Universal Robots PolyScope program: CameraCalibrate.urp

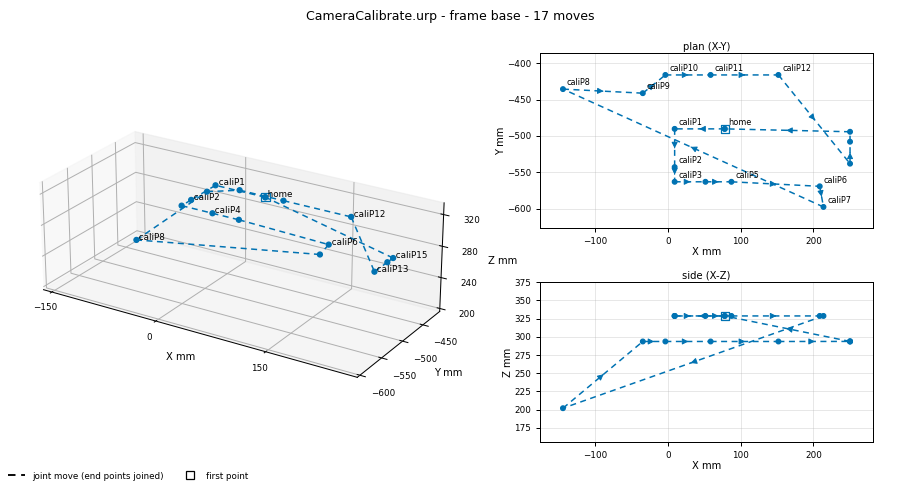
[picture p0: tool path of CameraCalibrate.urp in frame base, 17 of 17 moves have a stored position in this frame; points joined in program order, loops and branches not executed]
Program CameraCalibrate (installation=default directory=/programs/cam createdIn=5.19.0 lastSavedIn=5.15.1 robotSerialNumber=20245500285)
Calibrated DH parameters: a=[0.000097, -0.210459, -0.026602, 0.000137, 0.000078, 0]; d=[0.162601, 254.180657, -54.076236, -199.970743, 0.099615, 0.099684]; alpha=[1.569796, -0.001455, 0.001957, 1.570525, -1.571561, 0]; deltaTheta=[0, -1.053331, 8.839472, -1.50296, 0.000002, 0]
InitVariablesNode
Robot Program (runOnlyOnce=true)
  Script file /programs/cam/camera.script
    | def CameraOpenSock(ip, port=8888):
    |   socket_open(ip, port, "socker_camera")
    | end
    | 
    | 
    | def CameraCloseSock():
    |   socket_close("socker_camera")
    | end
    | 
    | 
    | def CameraSwitchOnline():
    |   socket_send_string("2\r", "socker_camera")
    |   ret = socket_read_string("socker_camera", suffix="\r")
    |   if (ret == "-1"):
    |     popup("CameraSwitchOnline Error", title="2.5D Camera", blocking=True)
    |   elif (ret == ""):
    |     popup("CameraSwitchOnline Error | Recv Data is None", title="2.5D Camera", blocking=True)
    |   end
    | end
    | 
    | 
    | def CameraStartCalibrate():
    |   socket_send_string("3\r", "socker_camera")
    |   ret = socket_read_string("socker_camera", suffix="\r")
    |   if (ret == "-1"):
    |     popup("CameraStartCalibrate Error", title="2.5D Camera", blocking=True)
    |   elif (ret == ""):
    |     popup("CameraStartCalibrate Error | Recv Data is None", title="2.5D Camera", blocking=True)
    |   end
    | end
    | 
    | def format03f(num):
    |   s = to_str(num)
    |   index = str_find(s, ".")
    |   if index != -1:
    |     ret = str_sub(s,0, index + 3)
    |     return ret
    |   else:
    |     return "rt"
    |   end
    | end
    | 
    | def CameraPackPose(pose):
    |   ret = ["", "", "", "", "", ""]
    |   pose[0] = pose[0] * 1000
    |   pose[1] = pose[1] * 1000
    |   pose[2] = pose[2] * 1000
    |   rpy = rotvec2rpy([pose[3], pose[4], pose[5]])
    |   ret[0] = format03f(pose[0])
    |   ret[1] = format03f(pose[1])
    |   ret[2] = format03f(pose[2])
    |   ret[3] = format03f(r2d(rpy[0]))
    |   ret[4] = format03f(r2d(rpy[1]))
    |   ret[5] = format03f(r2d(rpy[2]))
    |   i = 0
    |   out = ""
    |   while i < 6:
    |     out = str_cat(str_cat(out, ret[i]), ",")
    |     i = i + 1
    |   end
    | 
    |   return out
    | end
    | 
    | def CameraUnpackPose(text):
    |   ret = [0, 0, 0, 0, 0, 0, 0]
    |   i = 0
    |   index = 1
    |   while 1:
    |     index = str_find(text, ",")
    |     if index == -1:
    |       ret[i] = to_num(str_sub(text, 0))
    |     else:
    |       ret[i] = to_num(str_sub(text, 0, index))
    |     end
    |     text = str_sub(text, index+1)
    |     i=i+1
    |     if i > 6:
    |       break
    |     end
    |   end
    |   return ret
    | end
    | 
    | def CameraCalibrate(pose, num):
    | 
    |   pose1 = CameraPackPose(pose)
    |   sendStr = str_cat("", pose1)
    |   sendStr = str_cat("4,", sendStr)
    |   sendStr = str_cat(sendStr, to_str(num))
    |   sendStr = str_cat(sendStr, "\r")
    |   socket_send_string(sendStr, "socker_camera")
    |   ret = socket_read_string("socker_camera", suffix="\r")
    |   if (ret == "-1"):
    |     popup("CameraCalibrate Error", title="2.5D Camera", blocking=True)
    |   elif (ret == ""):
    |     popup("CameraCalibrate Error | Recv Data is None", title="2.5D Camera", blocking=True)
    |   end
    | end
    | 
    | 
    | def CameraEndCalibrate():
    |   socket_send_string("5\r", "socker_camera")
    |   ret = socket_read_string("socker_camera", suffix="\r")
    |   if (ret == "-1"):
    |     popup("CameraEndCalibrate Error", title="2.5D Camera", blocking=True)
    |   elif (ret == ""):
    |     popup("CameraEndCalibrate Error | Recv Data is None", title="2.5D Camera", blocking=True)
    |   end
    | end
    | 
    | 
    | def CameraGetCalibrateResult():
    | 
    |   socket_send_string("6\r")
    |   ret = socket_read_string("socker_camera", suffix="\r")
    |   if (ret == "-1"):
    |     popup("CameraGetCalibrateResult Error", title="2.5D Camera", blocking=True)
    |   elif (ret == ""):
    |     popup("CameraGetCalibrateResult Error | Recv Data is None", title="2.5D Camera", blocking=True)
    |   end
    | end
    | 
    | def CameraGetMarkPose():
    |   socket_send_string("1\r")
    |   ret = socket_read_string("socker_camera", suffix="\r")
    |   if (ret == "-1"):
    |     popup("CameraGetMarkPose Error", title="2.5D Camera", blocking=True)
    |   elif (ret == ""):
    |     popup("CameraGetMarkPose Error | Recv Data is None", title="2.5D Camera", blocking=True)
    |   else:
    |     result = CameraUnpackPose(ret)
    |     x = result[1] / 1000
    |     y = result[2] / 1000
    |     z = result[3] / 1000
    |     rx = d2r(result[4])
    |     ry = d2r(result[5])
    |     rz = d2r(result[6])
    |     rotvec2rpy = rpy2rotvec([rx, ry, rz])
    |     return [x, y, z, rotvec2rpy[0], rotvec2rpy[1], rotvec2rpy[2]]
    |   end
    | end
    | 
    | 
    | def CameraSaveTemplate(boardPose, tool=get_actual_tcp_pose()):
    |   # global CameraTemplate
    |   CameraTemplate = pose_trans(tool, boardPose)
    |   return CameraTemplate
    | end
    | 
    | def CameraTrsf(t, nT, p, tool=get_actual_tcp_pose()):
    |   trsf = pose_trans(pose_inv(t), p)
    |   ret = pose_trans(nT, trsf)
    |   return ret
    | end
  Script: CameraOpenSock("192.168.1.99", 8888)
  Script: CameraStartCalibrate()
  MoveJ speed 60 deg/s, acceleration 80 deg/s^2 (useActiveTCP=true) feature=Base
    Waypoint home: TCP in base x=78.162 y=-490.219 z=328.716 mm, rx=1.953 ry=2.4607 rz=0 rad; joints [83.356, -87.304, 111.233, -113.971, -90.025, 70.396] deg
    Script: CameraCalibrate(get_actual_tcp_pose(),1)
  MoveJ speed 60 deg/s, acceleration 80 deg/s^2 (useActiveTCP=true) feature=Base
    Waypoint caliP1: TCP in base x=9.395 y=-490.216 z=328.711 mm, rx=1.8055 ry=2.275 rz=0.262 rad; joints [71.893, -88.338, 111.523, -108.01, -74.336, 58.227] deg
    Script: CameraCalibrate(get_actual_tcp_pose(),2)
    Waypoint caliP2: TCP in base x=9.386 y=-542.747 z=328.724 mm, rx=1.8823 ry=2.3141 rz=0.4621 rad; joints [74.13, -79.525, 99.578, -96.524, -76.666, 60.977] deg
    Script: CameraCalibrate(get_actual_tcp_pose(),3)
    Waypoint caliP3: TCP in base x=9.395 y=-562.886 z=328.708 mm, rx=-1.9478 ry=-2.3477 rz=-0.4503 rad; joints [76.344, -75.67, 93.847, -91.652, -85.665, 65.265] deg
    Script: CameraCalibrate(get_actual_tcp_pose(),4)
    Waypoint caliP4: TCP in base x=51.659 y=-562.887 z=328.728 mm, rx=-1.9083 ry=-2.2531 rz=-0.2891 rad; joints [81.931, -75.392, 93.786, -93.635, -92.499, 72.966] deg
    Script: CameraCalibrate(get_actual_tcp_pose(),5)
    Waypoint caliP5: TCP in base x=87.316 y=-562.899 z=328.725 mm, rx=-1.8729 ry=-2.1767 rz=-0.1707 rad; joints [86.57, -74.564, 92.86, -93.637, -97.887, 79.191] deg
    Script: CameraCalibrate(get_actual_tcp_pose(),6)
    Waypoint caliP6: TCP in base x=208.594 y=-569.092 z=328.725 mm, rx=-1.7604 ry=-1.959 rz=0.1217 rad; joints [100.768, -67.818, 83.402, -84.689, -111.16, 98.788] deg
    Script: CameraCalibrate(get_actual_tcp_pose(),7)
    Waypoint caliP7: TCP in base x=213.728 y=-597.42 z=328.73 mm, rx=-1.7055 ry=-1.9272 rz=0.1003 rad; joints [100.941, -63.086, 76.071, -78.574, -112.507, 99.081] deg
    Script: CameraCalibrate(get_actual_tcp_pose(),8)
    Waypoint caliP8: TCP in base x=-143.969 y=-435.62 z=202.03 mm, rx=-0.4349 ry=2.6519 rz=0.5042 rad; joints [-95.138, -102.858, -115.737, -78.365, 106.879, -27.84] deg
    Script: CameraCalibrate(get_actual_tcp_pose(),9)
    Waypoint caliP9: TCP in base x=-34.347 y=-441.212 z=293.647 mm, rx=1.7983 ry=2.2001 rz=0.0566 rad; joints [63.83, -93.734, 124.614, -122.707, -72.812, 52.787] deg
    Script: CameraCalibrate(get_actual_tcp_pose(),10)
    Waypoint caliP10: TCP in base x=-3.351 y=-416.174 z=293.66 mm, rx=1.7423 ry=2.1705 rz=-0.1183 rad; joints [66.091, -98.263, 131.424, -133.489, -71.673, 55.418] deg
    Script: CameraCalibrate(get_actual_tcp_pose(),11)
    Waypoint caliP11: TCP in base x=58.77 y=-416.17 z=293.653 mm, rx=1.8028 ry=2.3259 rz=-0.352 rad; joints [78.661, -96.575, 131.561, -141.783, -87.034, 64.797] deg
    Script: CameraCalibrate(get_actual_tcp_pose(),12)
    Waypoint caliP12: TCP in base x=151.884 y=-416.164 z=293.638 mm, rx=-1.7862 ry=-2.419 rz=0.6473 rad; joints [96.807, -90.978, 126.971, -141.679, -109.249, 77.154] deg
    Script: CameraCalibrate(get_actual_tcp_pose(),13)
    Waypoint caliP13: TCP in base x=250.21 y=-538.008 z=293.739 mm, rx=-1.6396 ry=-2.0966 rz=0.2595 rad; joints [105.87, -68.815, 91.355, -96.275, -114.317, 95.631] deg
    Script: CameraCalibrate(get_actual_tcp_pose(),14)
    Waypoint caliP14: TCP in base x=250.21 y=-507.867 z=293.734 mm, rx=-1.7007 ry=-2.1157 rz=0.3788 rad; joints [106.958, -73.025, 98.472, -104.432, -115.782, 97.246] deg
    Script: CameraCalibrate(get_actual_tcp_pose(),15)
    Waypoint caliP15: TCP in base x=250.214 y=-494.194 z=293.719 mm, rx=-1.7394 ry=-2.1257 rz=0.4584 rad; joints [107.557, -74.946, 101.996, -109.5, -116.88, 98.117] deg
    Script: CameraCalibrate(get_actual_tcp_pose(),16)
  MoveJ speed 60 deg/s, acceleration 80 deg/s^2 (useActiveTCP=true) feature=Base
    Waypoint home: TCP in base x=78.162 y=-490.219 z=328.716 mm, rx=1.953 ry=2.4607 rz=0 rad; joints [83.356, -87.304, 111.233, -113.971, -90.025, 70.396] deg
    Script: CameraEndCalibrate()
    CameraTemplate := CameraSaveTemplate(CameraGetMarkPose())
  Script: CameraCloseSock()
